TYPE ST_SL_Steuerung :
STRUCT
	Freigabe		: ST_Steuerung_auto_manu_BOOL;
	Freigabe_Deakt	: ST_Steuerung_auto_manu_BOOL;

	Stellung_Anford	: ST_Steuerung_auto_manu_opti_BOOL; (*Wird hier nicht benötigt, sobald FB_SL_Logik angepasst wurde*)

	Ampel			: ST_Steuerung_auto_manu_opti_SINT; (*Hier lässt sich die Ampelfarbe wählen*)
	Blaue_Leuchte	: ST_Steuerung_auto_manu_opti_BOOL;	(*Ein und Ausschalten der blauen Leuchte*)
	Hupe			: ST_Steuerung_auto_manu_opti_BOOL; (*Ein und Ausschalten der Hupe*)

	Quittierung		: BOOL;
END_STRUCT
END_TYPE

(* stored: Version 1.1.0.1, ProductVersion 3.1.4024.9
   DUT ST_SL_Steuerung: Id {d88d6885-db50-4df7-888f-916a8f62b8ab} *)
